(* IEC 61131-3 sources: volt/packages/volt-lsp-iec/test-corpus/lenze-mid, 2 files *)

(* ---- GVL_Errorlists.gvl ---- *)
(* This code ist generated automatically *)
(* Don't change the content! *)

VAR_GLOBAL
	(* #7f7557b4-196d-4a0c-9db7-167ec53980dd# *)
	ATD_Errorlist : WORD:= 15360;
END_VAR
%LINK_ALWAYS

(* ---- POE_SystemStart.pou ---- *)
FUNCTION POE_SystemStart : DWORD
VAR_IN_OUT
	EventPrm: CmpApp.EVTPARAM_CmpApp;
END_VAR
VAR
END_VAR

%LANGUAGE LD
%NETWORK

END_FUNCTION
